//{attribute 'qualified_only'}
VAR_GLOBAL
END_VAR

(* stored: Version 1.1.0.1, ProductVersion 3.1.4024.12
   GVL GVL_SP1L0_Constants: Id {1190fd78-3e4f-42da-a68e-899711a263a1} *)
